// TIA Portal V20 export
TYPE "typeSafetyOperationEnable"
// stored: Access Published, IsFailsafeCompliant true, Namespace Safety
   STRUCT
      autoStartEnable : Bool;   // Auto Start Enable Status
      doorLockEnable : Bool;   // Door Lock Enable Status
      doorUnlockEnable : Bool;   // Door UnLock Enable Status
      rc_AutoEnable : Bool;   // Roll Change Auto Enable Status
      rc_RollChangeEnable : Bool;   // Roll Change Enable Status
      rc_DoorLockEnable : Bool;   // Roll Change Door Lock Enable Status
      rc_DoorUnlockEnable : Bool;   // Roll Change Door UnLock Enable Status
      hmiOperationEnable : Bool;   // Hmi Operation Enable Status with EnableBtn
      phmiOperationEnable : Bool;   // pHmi Operation Enable Status with EnableBtn
   END_STRUCT;
END_TYPE
